FUNCTION_BLOCK OctaOut_8_DO (* Service Interface Function Block Type *)
  (* Function: All Outputs; Description: Copyright (c) 2018, 2023 Jose Cabral, HR Agrartechnik GmbH This program and the accompanying materials are made available under the terms of the Eclipse Public License 2.0 which is available at https://www.eclipse.org/legal/epl-2.0/ SPDX-License-Identifier: EPL-2.0 this maps to QX *)
  (* Version 1.0, 2018-12-05, Jose Cabral *)
  (* Version 1.1, 2022-08-04, Franz Höpfinger, HR Agrartechnik GmbH *)
  (* Version 1.2, 2023-01-05, Franz Höpfinger, HR Agrartechnik GmbH *)
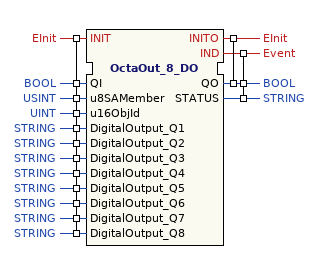
  EVENT_INPUT
    INIT : EInit WITH QI, u8SAMember, u16ObjId, DigitalOutput_Q1, DigitalOutput_Q2, DigitalOutput_Q3, DigitalOutput_Q4, DigitalOutput_Q5, DigitalOutput_Q6, DigitalOutput_Q7, DigitalOutput_Q8; (* Service Initialization *)
  END_EVENT
  EVENT_OUTPUT
    INITO : EInit WITH QO; (* Initialization Confirm *)
    IND WITH QO, STATUS; (* Indication from Resource *)
  END_EVENT
  VAR_INPUT
    QI : BOOL; (* Event Input Qualifier *)
    u8SAMember : USINT := isobus::GLOBAL; (* Dummy !, set to GLOBAL if in doubt. OFF deactivates FB. *)
    u16ObjId : UINT := isobus::ID_NULL; (* Dummy ! set to ID_NULL if in Doubt. ID_OFF deactivates FB. *)
    DigitalOutput_Q1 : STRING;
    DigitalOutput_Q2 : STRING;
    DigitalOutput_Q3 : STRING;
    DigitalOutput_Q4 : STRING;
    DigitalOutput_Q5 : STRING;
    DigitalOutput_Q6 : STRING;
    DigitalOutput_Q7 : STRING;
    DigitalOutput_Q8 : STRING;
  END_VAR
  VAR_OUTPUT
    QO : BOOL; (* Event Output Qualifier *)
    STATUS : STRING; (* Service Status *)
  END_VAR
END_FUNCTION_BLOCK
